{attribute 'linkalways'} 
{attribute 'no_explicit_call' := 'This FB is a CLASS and must be accessed using methods or properties'}
{attribute 'enable_dynamic_creation'}
FUNCTION_BLOCK FINAL Node_NOR EXTENDS Node
VAR
	in1 : _BOOL(FALSE);
    in2 : _BOOL(FALSE);
	out : _BOOL(FALSE);
END_VAR

METHOD PUBLIC  Clone : I_Node
VAR
	pNode : POINTER TO Node_NOR;
END_VAR
pNode := __NEW(Node_NOR);
Clone := pNode^;
END_METHOD

METHOD FB_init : BOOL
VAR_INPUT
	bInitRetains : BOOL; // if TRUE, the retain variables are initialized (warm start / cold start)
	bInCopyCode : BOOL;  // if TRUE, the instance afterwards gets moved into the copy code (online change)
END_VAR
AddParameter('in1', in1);
AddParameter('in2', in2);
AddOutput('out', out);

this^.Metadatum.AddBoolAsMetadata('deprecated', true);
END_METHOD

METHOD PROTECTED OnExecute
VAR
END_VAR
out.Value := NOT(in1.Value OR in2.Value);
END_METHOD

END_FUNCTION_BLOCK

(* stored: Version 1.1.0.1, ProductVersion 3.1.4026.18
   POU Node_NOR: Id {6c3559b6-bfca-05f9-0b5c-635fa7e8552f}, SpecialFunc None
   Folder Constructor: Id {37008843-bb28-0d14-1b7f-d64bfded3a11}
   Method Clone: Id {35ae8e80-bb89-0f8f-34b8-545255b7b624}
   Method FB_init: Id {7b82f80e-810f-0456-271e-ff666a43889f}
   Method OnExecute: Id {8eff7014-f701-0265-1b20-7a05e4f59099} *)
